TYPE ST_GCodeInfo :
STRUCT
	nNciState	: UDINT;
	nFileNr		: UDINT;
	nFileOffset : UDINT;
	nCurrentObj	: UINT;
	eGCodeState : E_GCodeState;
END_STRUCT
END_TYPE

(* stored: Version 1.1.0.1, ProductVersion 3.1.4020.12
   DUT ST_GCodeInfo: Id {80411860-89de-44fd-83d3-b800c09cac04} *)
